% RSLogix 500 project I2A-Job 18-Mitch.RSS, saved by version 10.00.00.00 %
PROJECT "ML01B"    % processor: Bul.1763 MicroLogix 1100 Series B %

PROGRAM FILES
  LAD 2   11 rungs

DATA FILES
  O0 OUTPUT  4 elements
  I1 INPUT  6 elements
  S2 STATUS  66 elements
  B3 BINARY  1 elements
  T4 TIMER  1 elements
  C5 COUNTER  1 elements
  R6 CONTROL  1 elements
  N7 INTEGER  1 elements
  F8 FLOAT  1 elements

LADDER 2
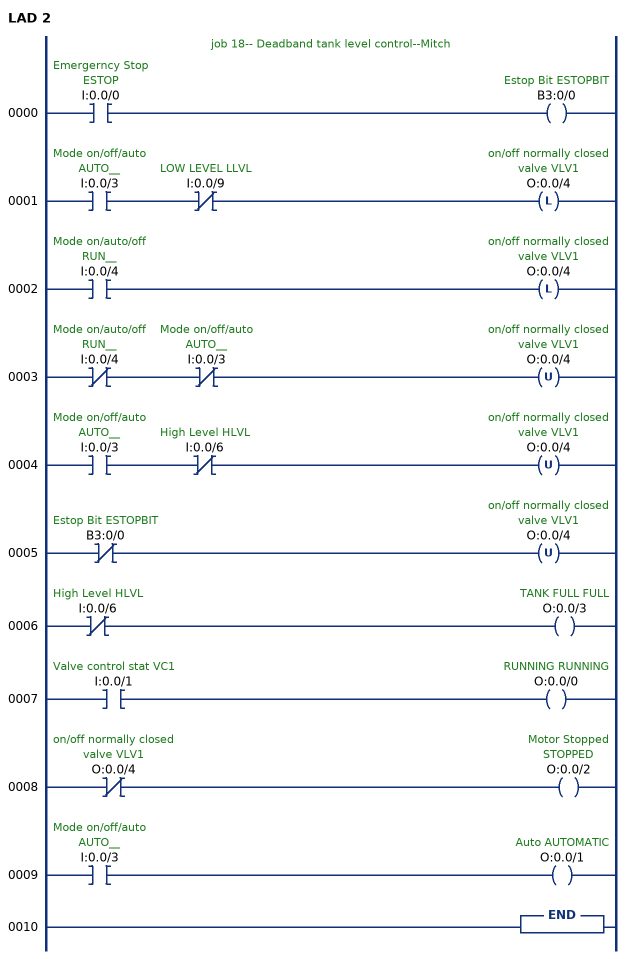
% Rung: 0 %
% job 18-- Deadband tank level control--Mitch %
SOR XIC I:0.0/0 OTE B3:0/0 EOR
%   I:0.0/0  ESTOP  "Emergerncy Stop" %
%   B3:0/0  ESTOPBIT  "Estop Bit" %
% Rung: 1 %
SOR XIC I:0.0/3 XIO I:0.0/9 OTL O:0.0/4 EOR
%   I:0.0/3  AUTO__  "Mode on/off/auto" %
%   I:0.0/9  LLVL  "LOW LEVEL" %
%   O:0.0/4  VLV1  "on/off normally closed valve" %
% Rung: 2 %
SOR XIC I:0.0/4 OTL O:0.0/4 EOR
%   I:0.0/4  RUN__  "Mode on/auto/off" %
%   O:0.0/4  VLV1  "on/off normally closed valve" %
% Rung: 3 %
SOR XIO I:0.0/4 XIO I:0.0/3 OTU O:0.0/4 EOR
%   I:0.0/4  RUN__  "Mode on/auto/off" %
%   I:0.0/3  AUTO__  "Mode on/off/auto" %
%   O:0.0/4  VLV1  "on/off normally closed valve" %
% Rung: 4 %
SOR XIC I:0.0/3 XIO I:0.0/6 OTU O:0.0/4 EOR
%   I:0.0/3  AUTO__  "Mode on/off/auto" %
%   I:0.0/6  HLVL  "High Level" %
%   O:0.0/4  VLV1  "on/off normally closed valve" %
% Rung: 5 %
SOR XIO B3:0/0 OTU O:0.0/4 EOR
%   B3:0/0  ESTOPBIT  "Estop Bit" %
%   O:0.0/4  VLV1  "on/off normally closed valve" %
% Rung: 6 %
SOR XIO I:0.0/6 OTE O:0.0/3 EOR
%   I:0.0/6  HLVL  "High Level" %
%   O:0.0/3  FULL  "TANK FULL" %
% Rung: 7 %
SOR XIC I:0.0/1 OTE O:0.0/0 EOR
%   I:0.0/1  VC1  "Valve control stat" %
%   O:0.0/0  RUNNING  "RUNNING" %
% Rung: 8 %
SOR XIO O:0.0/4 OTE O:0.0/2 EOR
%   O:0.0/4  VLV1  "on/off normally closed valve" %
%   O:0.0/2  STOPPED  "Motor Stopped" %
% Rung: 9 %
SOR XIC I:0.0/3 OTE O:0.0/1 EOR
%   I:0.0/3  AUTO__  "Mode on/off/auto" %
%   O:0.0/1  AUTOMATIC  "Auto" %
% Rung: 10 %
SOR END EOR

OTHER DOCUMENTED ADDRESSES
  B3:0/1  FWDB  "FWD BIT"
  B3:0/2  REVBIT  "REV BIT"
  B3:0/3  LAST_FWD  "LAST Forward"
  B3:0/4  LAST_REV  "Last Reverse"
  B3:0/5  RUN  "RUn Bit"
  B3:0/6  FJOG  "FWD Jog"
  B3:0/7  RJOG  "Rev Jog"
  B3:0/8  LATCH1  "LATCH"
  B3:0/9  UNLATCH  "Unlatch"
  I:0.0/2  MDR_STAT  "Motor Direction Contacts"
  I:0.0/5  AUTO  "OFF OR AUTO"
  I:0.0/7  START  "Start Motor"
  I:0.0/8  JOG  "Jog Motor"
  O:0.0/5  CR2ST  "Control relay 2"
  T4:0  MTR_TMR  "Motor Timer"
  T4:0/DN  T4
  T4:0/TT  TTT
  T4:1/TT  TT

DATA TABLE (non-zero values as saved)
DATA B3
% B3:0 % 0X0101
DATA T4
% .PRE .ACC %
% T4:0 % 32767 0
DATA C5
% .PRE .ACC %
% C5:0 % 16 0
